// TwinCAT 3 PLC project TFM
// ProgramVersion: 3.1.4024.0
// libraries:
//   Tc2_Standard, * (Beckhoff Automation GmbH)
//   Tc2_System, * (Beckhoff Automation GmbH)
//   Tc3_Module, * (Beckhoff Automation GmbH)
// project tree:
//   GVLs/ GVL_Inputs.TcGVL, GVL_Outputs.TcGVL
//   / PlcTask.TcTTO
//   POUs/ MAIN.TcPOU
// real-time tasks:
//   TASK PlcTask: cycle T#10ms, priority 20, ADS port 350

CONFIGURATION TFM
    RESOURCE PLC ON TwinCAT3
        TASK PlcTask(INTERVAL := T#10ms, PRIORITY := 20);
        PROGRAM MAIN WITH PlcTask : MAIN;
    END_RESOURCE
END_CONFIGURATION

// ---- GVLs/GVL_Inputs.TcGVL
{attribute 'qualified_only'}
VAR_GLOBAL

	{attribute 'OPC.UA.DA' := '1'}
	bStart  : BOOL; // Boton de start cuadro
	
	{attribute 'OPC.UA.DA' := '1'}
	bStop  : BOOL; // Boton de stop cuadro
	
	{attribute 'OPC.UA.DA' := '1'}
    setaEmergencia  : BOOL; // Seta emergencia cuadro

    {attribute 'OPC.UA.DA' := '1'}
	sensorDifuso1 : BOOL; // Sensor difuso 1

	{attribute 'OPC.UA.DA' := '1'}
	sensorDifuso2 : BOOL; // Sensor difuso 2
	
	{attribute 'OPC.UA.DA' := '1'}
	sensorDifus3 : BOOL; // Sensor difuso 3
	
	{attribute 'OPC.UA.DA' := '1'}
	sensorDifuso4 : BOOL; // Sensor difuso 4
	
	
END_VAR

VAR_GLOBAL CONSTANT
	
	//numero de sensores
    numSensores : INT := 4;
	

END_VAR

// ---- GVLs/GVL_Outputs.TcGVL
{attribute 'qualified_only'}
VAR_GLOBAL
	
	
	//numero de cintas
	//numCintas : INT;
	
	{attribute 'OPC.UA.DA' := '1'}
	luzVerdeCuadro : BOOL; // Senal luminosa verde cuadro 
	
	{attribute 'OPC.UA.DA' := '1'}
	luzAmarillaCuadro : BOOL; // Senal luminosa amarilla cuadro 

	{attribute 'OPC.UA.DA' := '1'}
	luzRojaCuadro : BOOL; // Senal luminosa roja cuadro 
	
	{attribute 'OPC.UA.DA' := '1'}
	cinta1 : BOOL; // cinta emisora bases

	{attribute 'OPC.UA.DA' := '1'}
	cinta2 : BOOL; // cinta 2 
	
	{attribute 'OPC.UA.DA' := '1'}
	cinta3 : BOOL; // cinta 3
	
	{attribute 'OPC.UA.DA' := '1'}
	cintaSalidaColor : BOOL; // cinta descarte por color 
	
END_VAR



VAR_GLOBAL CONSTANT
	
	
	//numero de cintas
	numCintas : INT := 4;

END_VAR

// ---- POUs/MAIN.TcPOU
PROGRAM MAIN
VAR
	
	enclaveCinta1 : BOOL; // Realimentacion boton start
	
	encendidoCinta1 : BOOL;
	encendidoCinta2 : BOOL;
	encendidoCinta3 : BOOL;
	encendidoCintaSalidaColor : BOOL;
	
    cintas : ARRAY[0..GVL_Outputs.numCintas] OF BOOL;
	sensores: ARRAY[0..GVL_Inputs.numSensores] OF BOOL;

	
	i: INT;// Indice contador
	//fBajada : ARRAY[0..GVL_Inputs.numSensores] OF F_TRIG;
	fBajada0 : F_TRIG;
	
	
	
END_VAR

VAR_INPUT
	enclaveCinta2: BOOL;
END_VAR

(*Si se acciona el boton de start 
se arranca la cinta de emision*)
IF GVL_Inputs.bStart THEN
	
	enclaveCinta1 := TRUE ; // Se mantiene la accion de start
	
END_IF



IF enclaveCinta1 THEN
	cintas[0] :=TRUE;
	
	// Arrancar segudanda cinta 
	//si el sensor del final de la cinta 1 detecta elemento
	IF GVL_Inputs.sensorDifuso1 THEN
//		cintas[1] := TRUE;
		enclaveCinta2 := TRUE;
	END_IF
	
	//Parar cinta 1 POR FLANCO
	fBajada0(CLK:= GVL_Inputs.sensorDifuso1);
	IF fBajada0.Q THEN
		cintas[0] := FALSE;
	END_IF
	
	// Parar cinta y comprobar color 
	// Arrancar cinta y orientar rodillos	
	
	
END_IF

IF enclaveCinta2 THEN
	cintas[1] := TRUE;
END_IF

//// Se paran todas las cintas y estaciones
IF  NOT GVL_Inputs.bStop THEN
	
	//Se paran todas las cintas
	FOR i := 0 TO GVL_Outputs.numCintas DO
		cintas[i] := FALSE;
	END_FOR
//	cintas[0] := FALSE;
//	cintas[1] := FALSE;
	enclaveCinta1 := FALSE;
	enclaveCinta2 := FALSE;
	
	// Se paran las estaciones (paletizado, montaje final etc)
	
END_IF


//Actualizar salidas
GVL_Outputs.cinta1 := cintas[0];
GVL_Outputs.cinta2 := cintas[1];
GVL_Outputs.cinta3 := cintas[2];
GVL_Outputs.cintaSalidaColor := cintas[3];

END_PROGRAM
